FUNCTION_BLOCK FB_XpParallel
VAR_INPUT
END_VAR
VAR_OUTPUT
END_VAR
VAR
END_VAR

END_FUNCTION_BLOCK

(* stored: Version 1.1.0.1
   POU FB_XpParallel: Id {223e9b2d-4978-44f7-9960-9e033825c055}, SpecialFunc None *)
